(* IEC 61131-3 sources: repolevel_ST_code_completion/output/0122完整版本_无planner目前sota/repoeval_Builder_Application_RPI/readful_result_no_provide, 5 files *)

(* ---- Director.st ---- *)
{attribute 'enable_dynamic_creation'}
//The director class is responsible to delegate the construction of the final product object
// to a concrete builder object.
FUNCTION_BLOCK Director
VAR_INPUT
  //Reference to the builder that is going to be building the final product object.
  inputConcreteBuilder : ConcreteBuilder;
END_VAR
VAR_OUTPUT
END_VAR
VAR
  //Holds a reference to the concrete builder object to send the specifications of the final product to it.
  concreteBuilder : ConcreteBuilder;
END_VAR

//Stores the reference to which builder will be building the final product object in its own field THIS^.concreteBuilder
concreteBuilder := inputConcreteBuilder; // Removed the `THIS^.` prefix since it's unnecessary in a FUNCTION_BLOCK for accessing local variables

//The Director tells its concreteBuilder instance to build the final product step by step passing the specifications stored in the
// concreteBuilder array THIS^.specifications[1..4]

//Step 1 "Main Part"
IF concreteBuilder.specifications[1] >= 0 THEN // Adjusted condition to ensure compatibility with valid numeric comparisons
 concreteBuilder.Set_Main_Part(concreteBuilder.specifications[1]);
END_IF
//Step 2 "Part 1"
IF concreteBuilder.specifications[2] >= 0 THEN // Adjusted condition to ensure compatibility with valid numeric comparisons
 concreteBuilder.Set_Part1(concreteBuilder.specifications[2]);
END_IF
//Step 3 "Part 2"
IF concreteBuilder.specifications[3] >= 0 THEN // Adjusted condition to ensure compatibility with valid numeric comparisons
 concreteBuilder.Set_Part2(concreteBuilder.specifications[3]);
END_IF
//Step 4 "Part 3"
IF concreteBuilder.specifications[4] >= 0 THEN // Adjusted condition to ensure compatibility with valid numeric comparisons
 concreteBuilder.Set_Part3(concreteBuilder.specifications[4]);
END_IF

//Finally the concreteBuilder instance in the Director object delivers the final result as a Product object
concreteBuilder.Get_Result(); // Removed `THIS^.` prefix to match the local variable context of the FUNCTION_BLOCK
END_FUNCTION_BLOCK

(* ---- ConcreteBuilder.st ---- *)
VAR
  // Internal variables for building the product
  localProduct : Product; // Ensure 'Product' is a valid data type or function block
  specifications : ARRAY [1..4] OF STRING;
END_VAR

METHOD Set_Main_Part : BOOL // Removed erroneous VAR sections from method declarations
VAR_INPUT
  mainPart : STRING;
END_VAR
IF mainPart <> '' THEN
  localProduct.mainPart := mainPart;
  RETURN TRUE;
ELSE
  RETURN FALSE;
END_IF

METHOD Set_Part1 : BOOL // Removed erroneous VAR sections from method declarations
VAR_INPUT
  part1 : STRING;
END_VAR
IF part1 <> '' THEN
  localProduct.part1 := part1;
  RETURN TRUE;
ELSE
  RETURN FALSE;
END_IF

METHOD Set_Part2 : BOOL // Removed erroneous VAR sections from method declarations
VAR_INPUT
  part2 : STRING;
END_VAR
IF part2 <> '' THEN
  localProduct.part2 := part2;
  RETURN TRUE;
ELSE
  RETURN FALSE;
END_IF

METHOD Set_Part3 : BOOL // Removed erroneous VAR sections from method declarations
VAR_INPUT
  part3 : STRING;
END_VAR
IF part3 <> '' THEN
  localProduct.part3 := part3;
  RETURN TRUE;
ELSE
  RETURN FALSE;
END_IF

METHOD Reset : BOOL
localProduct := (mainPart := '', part1 := '', part2 := '', part3 := ''); // Ensure initializer is valid for 'localProduct'
RETURN TRUE;

END_FUNCTION_BLOCK

(* ---- Director_Construct.st ---- *)
VAR
	//Holds a reference to the concrete builder object to send the specifications of the final product to it.
	concreteBuilder : ConcreteBuilder(specs := THIS^.inputConcreteBuilder.specifications);
END_VAR

//Step 1 "Main Part"
concreteBuilder.Set_Main_Part(concreteBuilder.specifications[1]);
//Step 2 "Part 1"
concreteBuilder.Set_Part1(concreteBuilder.specifications[2]);
//Step 3 "Part 2"
concreteBuilder.Set_Part2(concreteBuilder.specifications[3]);
//Step 4 "Part 3"
concreteBuilder.Set_Part3(concreteBuilder.specifications[4]);

//Finally the concreteBuilder instance delivers the final result as a Product object
Construct := concreteBuilder.Get_Result();
RETURN;
END_OTHER

(* ---- Product.st ---- *)
VAR
// Index variable for iteration
  i : INT;
END_VAR

// Static initialization of parts as dynamic assignment is not possible without specifications
CASE i OF
  1: mainPart := 'DefaultMainPart'; // Set to static/default value
  2: part1 := 'DefaultPart1';      // Set to static/default value
  3: part2 := 'DefaultPart2';      // Set to static/default value
  4: part3 := 'DefaultPart3';      // Set to static/default value
END_CASE;
END_FUNCTION_BLOCK

(* ---- Product_toString.st ---- *)
VAR
    //Local variable to join together and store the pieces of String
    tempString: STRING;
END_VAR

//Concatenate "mainPart" and "part1"
tempString := CONCAT(mainPart, part1);
//Concatenate the current value of "tempString" with "part2"
tempString := CONCAT(tempString, part2);
//Concatenate the current value of "tempString" with "part3"
tempString := CONCAT(tempString, part3);
//Return the final concatenated string
toString := tempString;
RETURN;
END_OTHER
